Fanuc KAREL source: NC0081.KL

-- PROVISIONAL review KL for V1013-1; original PC SHA256 95f85d55a3ddde44e27eeb7ee8769af35fa1294229a21d2799cdcf10973b55d2
-- Incomplete behavior may be omitted. Consult companion uncertainty JSON. Do not deploy.
PROGRAM NC0081
%NOLOCKGROUP
-- UNRESOLVED_LOCAL_POOL 1 cells at code offset 3; source declarations unknown
-- DIRECT_LOCAL_WORD_ACCESS alone does not prove INTEGER, REAL, or BOOLEAN
BEGIN
  -- UNRESOLVED_PC offsets 0-8; opcodes 2B,2C,7B
  -- UNRESOLVED_PC offsets 13-20; opcodes 9D,23
  -- UNRESOLVED_PC offsets 25-42; opcodes 21,2E,59,79
  -- UNRESOLVED_PC offsets 47-64; opcodes 21,2E,59,79
  -- UNRESOLVED_PC offsets 69-86; opcodes 21,2E,59,79
  -- UNRESOLVED_PC offsets 91-108; opcodes 21,2E,59,79
  -- UNRESOLVED_PC offsets 113-130; opcodes 21,2E,59,79
  -- UNRESOLVED_PC offsets 135-152; opcodes 21,2E,59,79
  -- UNRESOLVED_PC offsets 157-174; opcodes 21,2E,59,79
  -- UNRESOLVED_PC offsets 179-196; opcodes 21,2E,59,79
  -- UNRESOLVED_PC offsets 201-218; opcodes 21,2E,59,79
  -- UNRESOLVED_PC offsets 223-240; opcodes 21,2E,59,79
  -- UNRESOLVED_PC offsets 245-262; opcodes 21,2E,59,79
  -- UNRESOLVED_PC offsets 267-284; opcodes 21,2E,59,79
  -- UNRESOLVED_PC offsets 289-306; opcodes 21,2E,59,79
  -- UNRESOLVED_PC offsets 311-328; opcodes 21,2E,59,79
  -- UNRESOLVED_PC offsets 333-350; opcodes 21,2E,59,79
  -- UNRESOLVED_PC offsets 355-372; opcodes 21,2E,59,79
  -- UNRESOLVED_PC offsets 377-394; opcodes 21,2E,59,79
  -- UNRESOLVED_PC offsets 399-416; opcodes 21,2E,59,79
  -- UNRESOLVED_PC offsets 421-438; opcodes 21,2E,59,79
  -- UNRESOLVED_PC offsets 443-460; opcodes 21,2E,59,79
  -- UNRESOLVED_PC offsets 465-479; opcodes 21,9D,52,23
  -- UNRESOLVED_PC offsets 484-489; opcodes 7A
  -- UNRESOLVED_PC offsets 494-499; opcodes 7A
  -- UNRESOLVED_PC offsets 504-509; opcodes 7A
  -- UNRESOLVED_PC offsets 514-519; opcodes 7A
  -- UNRESOLVED_PC offsets 524-529; opcodes 7A
  -- UNRESOLVED_PC offsets 534-539; opcodes 7A
  -- UNRESOLVED_PC offsets 544-549; opcodes 7A
  -- UNRESOLVED_PC offsets 554-559; opcodes 7A
  -- UNRESOLVED_PC offsets 564-569; opcodes 7A
  -- UNRESOLVED_PC offsets 574-579; opcodes 7A
  -- UNRESOLVED_PC offsets 584-589; opcodes 7A
  -- UNRESOLVED_PC offsets 594-599; opcodes 7A
  -- UNRESOLVED_PC offsets 604-609; opcodes 7A
  -- UNRESOLVED_PC offsets 614-619; opcodes 7A
  -- UNRESOLVED_PC offsets 624-629; opcodes 7A
  -- UNRESOLVED_PC offsets 634-639; opcodes 7A
  -- UNRESOLVED_PC offsets 644-649; opcodes 7A
  -- UNRESOLVED_PC offsets 654-659; opcodes 7A
  -- UNRESOLVED_PC offsets 664-669; opcodes 7A
  -- UNRESOLVED_PC offsets 674-679; opcodes 7A
  -- UNRESOLVED_PC offsets 684-688; opcodes 7F
  -- UNRESOLVED_PC offsets 693-697; opcodes 27,AA
  -- UNRESOLVED_PC offsets 702-706; opcodes 7F
END NC0081
